(* IEC 61131-3 sources: test/Class/HmiTextList35Manager, 1 file *)

(* ---- HmiTextList35Manager.st ---- *)
(*!
<Class
	Name               = "HmiTextList35Manager"
	Revision           = "0.0"
	RealtimeTask       = "false"
	CyclicTask         = "false"
	BackgroundTask     = "false"
	Sigmatek           = "true"
	OSInterface        = "false"
	HighPriority       = "false"
	Automatic          = "false"
	UpdateMode         = "Prescan"
	SharedCommandTable = "true"
	Objectsize         = "(284,120)">
	<Channels>
		<Server Name="ClassSvr" Visualized="false" Initialize="false" WriteProtected="true" Retentive="false"/>
	</Channels>
</Class>
*)
HmiTextList35Manager : CLASS
  //Servers:
	ClassSvr 	: SvrChCmd_DINT;
  //Clients:
  //Variables:
		xOffset : ARRAY [0..10000] OF UDINT;

  //Functions:

	FUNCTION GLOBAL SeekText
		VAR_INPUT
			list 	: ^UINT;
			no 	: UDINT;
			txt 	: ^UINT;
			length 	: UDINT;
		END_VAR
		VAR_OUTPUT
			retcode 	: UDINT;
		END_VAR;

	FUNCTION GLOBAL AddOffset
		VAR_INPUT
			index 	: UDINT;
			offset 	: UDINT;
		END_VAR
		VAR_OUTPUT
			retcode 	: BOOL;
		END_VAR;

	FUNCTION GLOBAL Zero;
  //Tables:
	FUNCTION @STD
		VAR_OUTPUT
			ret_code	: CONFSTATES;
		END_VAR;
	FUNCTION GLOBAL TAB @CT_;
END_CLASS;

FUNCTION GLOBAL HmiTextList35Manager::Zero

  _memset(#xOffset[0], 0, sizeof(xOffset));

END_FUNCTION

FUNCTION GLOBAL HmiTextList35Manager::SeekText
	VAR_INPUT
		list 	: ^UINT;
		no 	: UDINT;
		txt 	: ^UINT;
		length 	: UDINT;
	END_VAR
	VAR_OUTPUT
		retcode 	: UDINT;
	END_VAR
  var
    ph : ^uint;
  end_var

  if((no > 0) & (list <> NIL) & (txt <> NIL)) then
    while(no) do
      no -= 1;
      ph := list + xOffset[no];
      if(ph^ = txt^) then
        if(_memcmp(ph, txt, length) = 0) then
          retcode := no;
          return;
        end_if;
      end_if;
    end_while;
  end_if;

  retcode := 16#FFFFFFFF;

END_FUNCTION

FUNCTION GLOBAL HmiTextList35Manager::AddOffset
	VAR_INPUT
		index 	: UDINT;
		offset 	: UDINT;
	END_VAR
	VAR_OUTPUT
		retcode 	: BOOL;
	END_VAR

  retcode := false;
  if(index < (sizeof(xOffset) / sizeof(xOffset[0]))) then
    xOffset[index] := offset;
    retcode := true;
  end_if;

END_FUNCTION
